(* Schneider Machine Expert - Basic project demo2_timer, file version 2.2.0.0 *)
(* CompanyInformations: WebSite=https://ics-cybersecurity.academy *)
(* ProjectInformations: Name=ICSJWG demo2, Description=Simple timer to demonstrate why controls must be implemented on the PLC and not only in the SCADA, and why timers must be verified *)
(* UserInformations: LastName=Arnaud, FirstName=SOULLIE, Email=asoullie@ics-cybersecurity.academy *)

HARDWARE
  Cpu 0: TM221ME16R/G
  EthernetConfiguration: NetworkName=M221, IpAllocationMode=FixedAddress, IpAddress=192.168.0.53, SubnetMask=255.255.255.0
  SerialLineConfiguration: Baud=Baud19200, Parity=ParityEven, DataBits=DataBits8, StopBits=StopBits1, PhysicalMedium=PhysicalMediumRs485, TransmissionMode=TransmissionModeModbusRtu, SlaveId=1, Addressing=SlaveAddressing
  MastTask: UsePeriodScanMode=false, PeriodScan=100
  FastTask: Period=255
  CpuBehavior: StartingMode=StartAsPreviousState, AutoSaveRamOnEeprom=true, WatchdogPeriod=250

SYMBOLS  (address, symbol, comment, settings)
  %M0       TIMER_START
  %M20      WASH_INTAKE
  %M23      BARREL_VALVE
  %M100     IO_FORCED
  %M101     INPUT_FORCED
  %M102     OUTPUT_FORCED
  %MW0      TIMER_DURATION
  %MW10     STILL_TEMP
  %MW11     STILL_LEVEL
  %MW12     CONDENSER_TEMP
  %MW13     BARREL_LEVEL
  %MW21     HEATER
  %MW22     COOLING_PUMP
  %MW100    BOOTLOADER_VERSION
  %MW101    COMMERCIAL_VERSION
  %MW102    FIRMWARE_V_PART1
  %MW103    FIRMWARE_V_PART2
  %MW104    APPLICATION_SIGNATURE
  %MW110    LAST_SCAN_TIME
  %TM0        [Preset=10, Base=OneSecond]

POU Timer
  (* SectionNumber=1 *)

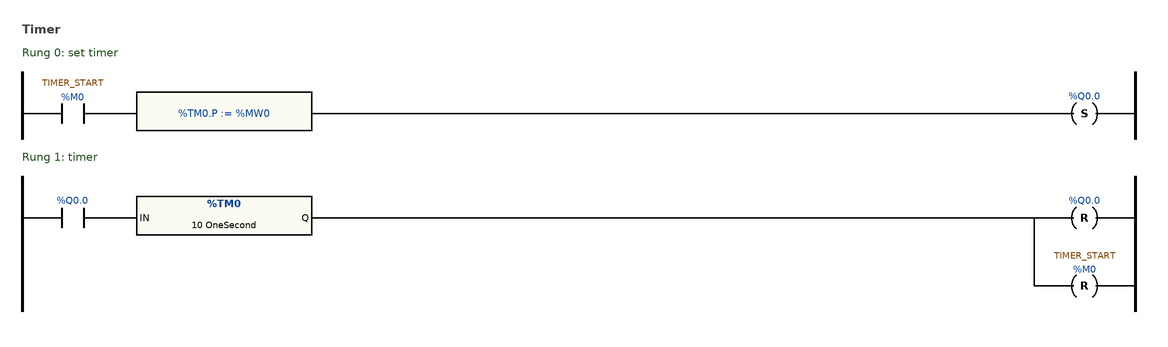

// Rung 0: set timer
  LD %M0                  (* TIMER_START *)
  OPER [ %TM0.P := %MW0 ] (* TIMER_DURATION *)
  S %Q0.0
  // as ST:
  //   IF TIMER_START THEN %TM0.P := TIMER_DURATION; END_IF;
  //   IF TIMER_START THEN %Q0.0 := TRUE; END_IF;

// Rung 1: timer
  BLK %TM0
  LD %Q0.0
  IN
  OUT_BLK
  LD Q
  R %Q0.0
  R %M0                   (* TIMER_START *)
  END_BLK
  // as ST:
  //   %TM0(IN := %Q0.0);
  //   IF %TM0.Q THEN %Q0.0 := FALSE; END_IF;
  //   IF %TM0.Q THEN TIMER_START := FALSE; END_IF;
